ADAPTER ISludgeBufferToReactors (* Adapter Interface *)
  (* Standard: 61499-1 *)
  (* Version 0.0, 9/17/2026, Schneider Electric *)
  PACKAGE SE.Nereda;
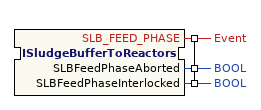
  EVENT_OUTPUT
    SLB_FEED_PHASE WITH SLBFeedPhaseAborted, SLBFeedPhaseInterlocked;
  END_EVENT
  VAR_OUTPUT
    SLBFeedPhaseAborted : BOOL;
    SLBFeedPhaseInterlocked : BOOL;
  END_VAR
  SERVICE SOCKET/PLUG
    SEQUENCE request_confirm
      SOCKET.REQ(REQD) -> PLUG.REQ(REQD);
      PLUG.CNF(ReactorFeedPhaseStarted) -> SOCKET.CNF(ReactorFeedPhaseStarted);
    END_SEQUENCE
    SEQUENCE indication_response
      PLUG.IND(INDD) -> SOCKET.IND(INDD);
      SOCKET.RSP(RSPD) -> PLUG.RSP(RSPD);
    END_SEQUENCE
  END_SERVICE
END_ADAPTER
